RoboDK station: DalsySinBD.rdk

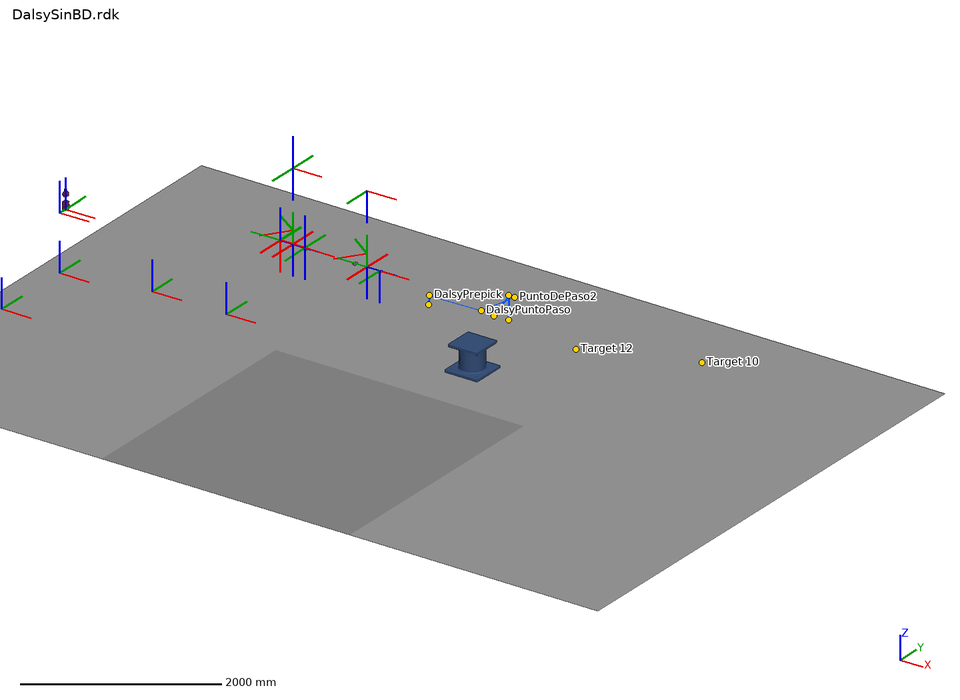
[picture v0: the station drawn from its stored meshes, robots at their saved joint values, targets as dots, program paths as lines]
Station EstacionProyectoFinaleliminarBotela (saved by RoboDK 5.9.4). Poses are relative to the parent item; angles as X-Y-Z fixed-axis rotations.
Station parameters (name, value as stored): Posicion, [[ 2850.000 ]] , CantBot1, 0, NUMBOTELLA1, 0, ElimBotellas1, 0, detectado1, 0, repes1, 0, Prellena1, 0, Prellena, 0, Detectado1, 0, IO_5, 1, NewPick, 0, Pinza, 1, NewPlace, 0, waituntil Detectado1, 1, Ventosa_plegado_caja, 0, CantCaja, 1.0, SCajaInicial, 1, SCajaPlace, 0, if(SCajaInicial, SyntaxError: Unexpected token `=', If(SCajaInicial, SyntaxError: Unexpected token `=', Mesa, 1, Mesa1, 0, Mesa2, 0, Mesa3, 0, MesaE, 0, MesaS, 1, Temperatura, 0, SensorMqtt, 0, LotesPendientes, 1
  - folder ESTACIÓN
    - folder Suelo
      - object Floor at (4500, 1500, 0) mm, size 3000 x 3000 x 0 mm, geometry from Floor.sld
      - object Floor2 at (1500, 1500, 0) mm, size 3000 x 3000 x 0 mm, geometry from Floor.sld
      - object Floor3 at (1500, 4500, 0) mm, size 3000 x 3000 x 0 mm, geometry from Floor.sld
      - object Floor4 at (4500, 4500, 0) mm, size 3000 x 3000 x 0 mm, geometry from Floor.sld
      - object Floor6 at (7500, 1500, 0) mm, size 3000 x 3000 x 0 mm, geometry from Floor.sld
      - object Floor5 at (7500, 4500, 0) mm, size 3000 x 3000 x 0 mm, geometry from Floor.sld
    - folder Mesa Giratoria
  - frame SisGeneral at (0, -19.13, 0) mm
    - folder CintayRobot
      - frame SisRefPick at (250, 2217.22, 0) mm
        - frame Cinta Botellas 1 at (0, 1000, 0) mm
          - robot CintaUno: 1 axes
              modified DH rows (alpha deg, a mm, theta deg, d mm): 0, 0, 0, 0 linear
              base shift (0, 0, 0) mm, rotated rx 0 ry 90 rz 0 deg
              joint limits [0] to [4500]; home [0]; saved at [0]
            - frame FrameBotellaSave at (0, 0, 0) mm
              - object Guardado at (0, 0, 0) mm, size 71.4 x 71.4 x 222.2 mm, 1042852009 curves, geometry from Bottle-Label.sld
            - frame Move at (0, 0, 0) mm
              - frame FrameBotella at (0, 100, 0) mm
                - object botella0 at (0, 0, 0) mm, size 71.4 x 71.4 x 222.2 mm, 1039516303 curves, geometry from Bottle-Label.sld
          - target Inicio (Cartesian target) at (0, 100, 863) mm; joints [0] of CintaUno
          - target Final (Cartesian target) at (4325.5, 559.3, 913.95) mm, rotated rx -90 ry 0 rz 90 deg; joints [0, -90, -90, 0, 90, 0] of CintaUno
          - frame TANQUE 1 at (1750, -902.14, 647.6) mm
            - frame Cono at (1000, 1000, 1240) mm, rotated rx 180 ry 0 rz 0 deg
              - object Cone 500x500mm at (0, 0, 0) mm
            - frame Deposito at (1000, 1000, 1240) mm
              - object Deposito at (0, 0, 0) mm
            - frame Frame 24 at (1000.71, 1000.6, 551.36) mm, rotated rx 180 ry 0 rz -124.91 deg
              - object Cylinder 50x150mm at (0, 0, 0) mm
            - frame Frame 25 at (1000.71, 1000.6, 401.36) mm, rotated rx -180 ry 0 rz -90 deg
              - object Cylinder 50x150mm at (0, 0, 0) mm
            - frame Frame 26 at (1000.71, 1000.6, 401.36) mm, rotated rx 90 ry 0 rz 90 deg
              - object Cylinder 50x150mm at (0, 0, 0) mm
            - frame Frame 27 at (1150.71, 1000.6, 401.36) mm, rotated rx -180 ry 0 rz 0 deg
              - object Cylinder 50x150mm at (0, 0, 0) mm
            - frame Frame 25 at (1000.71, 1000.6, 401.36) mm, rotated rx -180 ry 0 rz -90 deg
              - object Cylinder 50x150mm at (0, 0, 0) mm
            - frame Frame 25 at (850.71, 1000.6, 401.36) mm, rotated rx -180 ry 0 rz -90 deg
              - object Cylinder 50x150mm at (0, 0, 0) mm
            - frame Frame 25 at (850.71, 1000.6, 401.36) mm, rotated rx 0 ry 90 rz 0 deg
              - object Cylinder 50x150mm at (0, 0, 0) mm
            - frame Frame 31 at (850.65, 1001.38, 406.13) mm
              - object Sphere D100mm at (0, 0, 0) mm, size 50 x 50 x 25 mm, 1060155569 curves, geometry from Sphere-D100mm.sld
            - frame Frame 31 at (1151.57, 999.51, 402.52) mm
              - object Sphere D100mm at (0, 0, 0) mm, size 50 x 50 x 25 mm, 1060155569 curves, geometry from Sphere-D100mm.sld
          - frame DispensaTapones at (2650, -902.14, 647.6) mm
            - frame Cono at (1000, 1000, 1240) mm, rotated rx 180 ry 0 rz 0 deg
              - object Cone 500x500mm at (0, 0, 0) mm
            - frame Frame 24 at (1000.71, 1000.6, 551.36) mm, rotated rx 180 ry 0 rz -124.91 deg
              - object Cylinder 50x150mm at (0, 0, 0) mm
            - frame Frame 25 at (1000.71, 1000.6, 401.36) mm, rotated rx -180 ry 0 rz -90 deg
              - object Cylinder 50x150mm at (0, 0, 0) mm
            - frame Frame 26 at (1000.71, 1000.6, 401.36) mm, rotated rx 90 ry 0 rz 90 deg
              - object Cylinder 50x150mm at (0, 0, 0) mm
            - frame Frame 27 at (1150.71, 1000.6, 401.36) mm, rotated rx -180 ry 0 rz 0 deg
              - object Cylinder 50x150mm at (0, 0, 0) mm
            - frame Frame 25 at (1000.71, 1000.6, 401.36) mm, rotated rx -180 ry 0 rz -90 deg
              - object Cylinder 50x150mm at (0, 0, 0) mm
            - frame Frame 25 at (850.71, 1000.6, 401.36) mm, rotated rx -180 ry 0 rz -90 deg
              - object Cylinder 50x150mm at (0, 0, 0) mm
            - frame Frame 25 at (850.71, 1000.6, 401.36) mm, rotated rx 0 ry 90 rz 0 deg
              - object Cylinder 50x150mm at (0, 0, 0) mm
            - frame Frame 31 at (850.65, 1001.38, 406.13) mm
              - object Sphere D100mm at (0, 0, 0) mm, size 50 x 50 x 25 mm, 1060155569 curves, geometry from Sphere-D100mm.sld
            - frame Frame 31 at (1151.57, 999.51, 402.52) mm
              - object Sphere D100mm at (0, 0, 0) mm, size 50 x 50 x 25 mm, 1060155569 curves, geometry from Sphere-D100mm.sld
          - frame Sensor3 at (3498.8, -14.22, 715.35) mm, rotated rx 0 ry 0 rz 88.62 deg
            - object B2 at (0, 0, 0) mm
          - frame Sensor2 at (4402.28, -29.98, 715.35) mm, rotated rx 0 ry 0 rz 88.62 deg
            - object B1 at (0, 0, 0) mm
          - frame Sensor1 at (2598.8, -14.22, 715.35) mm, rotated rx 0 ry 0 rz 88.62 deg
            - object B0 at (0, 0, 0) mm
          - target DalsyPrepick (Cartesian target) at (4404.64, 97.25, 945.23) mm, rotated rx -179.46 ry -0.56 rz 92.6 deg; joints [67.794, -102.103, -28.32, -139.861, 89.279, 65.196] of UR5PickDalsy
          - target DalsyPick (Cartesian target) at (4400.29, 94.49, 846.14) mm, rotated rx -179.46 ry -0.56 rz 92.6 deg; joints [67.407, -90.716, -60.305, -119.258, 89.278, 64.809] of UR5PickDalsy
          - target DalsyPuntoPaso (Cartesian target) at (4989.54, 154.84, 921.17) mm, rotated rx 176.54 ry 3.78 rz 107.72 deg; joints [150.48, -91.95, -47.39, -125.54, 89.98, 132.65] of UR5PickDalsy
          - target PuntoDePaso2 (Cartesian target) at (5091.93, 592.06, 921.34) mm, rotated rx 176.53 ry 3.81 rz 169.24 deg; joints [212.01, -91.94, -47.38, -125.53, 89.97, 132.65] of UR5PickDalsy
          - target PrePlace (Cartesian target) at (5051.88, 544.46, 950.34) mm, rotated rx 179.87 ry 0 rz -95.46 deg; joints [208.979, -92.535, -38.825, -138.744, 90.075, 34.439] of UR5PickDalsy
          - target Place (Cartesian target) at (5051.88, 544.46, 680.34) mm, rotated rx 179.87 ry 0 rz -95.46 deg; joints [208.979, -74.687, -99.618, -95.799, 90.075, 34.439] of UR5PickDalsy
          - target Target 9 (Cartesian target) at (5079.28, 251.73, 846.24) mm, rotated rx -179.45 ry -0.55 rz -167.69 deg; joints [167.11, -90.71, -60.3, -119.25, 89.27, 64.8] of UR5PickDalsy
          - target Target 10 (Cartesian target) at (7103.35, 957.35, 614.14) mm, rotated rx -138.15 ry 89.07 rz -48.26 deg; joints [177.195, -131.024, -49.86, -164.778, 177.217, -76.295]
          - target Target 11 (Cartesian target) at (4404.64, 97.25, 945.23) mm, rotated rx -179.46 ry -0.56 rz 92.6 deg; joints [67.794, -102.103, -28.32, -139.861, 89.279, 65.196] of UR5PickDalsy
          - target Target 12 (Cartesian target) at (5875.13, 535.29, 591.77) mm, rotated rx -124.69 ry 88.93 rz 144.57 deg; joints [23.154, -118.729, -72.709, -170.068, 203.904, -92.258]
        - frame UR5 BasePickDalsy at (4673.46, 1459.5, 355) mm, rotated rx 0 ry 0 rz 180 deg
          - robot UR5PickDalsy (model UR5): 6 axes
              modified DH rows (alpha deg, a mm, theta deg, d mm): 0, 0, 0, 89.2; 90, 0, 180, 0; 0, 425, 0, 0; 0, 392, 0, 109.3; -90, 0, 0, 94.75; 90, 0, 180, 82.5
              joint limits [-360, -360, -360, -360, -360, -360] to [360, 360, 360, 360, 360, 360]; home [0, -90, -90, 0, 90, 0]; saved at [67.794, -102.103, -28.32, -139.861, 89.279, 65.196]
            - tool GripperPick, TCP at (0, 0, 130) mm
            - tool GripperPickV, TCP at (0, 0, 130) mm
          - frame Frame 45 at (4.13, 0, -300) mm
            - object Pedestal R1 at (0, 0, 0) mm, size 400 x 400 x 304.8 mm, 1065353216 curves, geometry from Pedestal-H12in-Type-1.sld
      - folder ProgramasDeLaCinta
        - Python program AvanzaCinta1 (listed below)
        - Python program AvanzaCinta2 (listed below)
        - Python program ResetBot (listed below)
        - program ProgCinta1 (11 instructions, listed below)
        - Python program ProgCintaUno (listed below)
      - folder Sensores
        - Python program ProgB0 (listed below)
        - Python program ProgB1 (listed below)
        - Python program ProgB2 (listed below)
      - folder ProgramasUr
        - program DalsyPickPlace (33 instructions, listed below)
        - Python program PickDalsy (listed below)
        - Python program PlaceDalsy (listed below)
        - Python program BorrarBotella (listed below)
    - folder Mesa
      - frame MesaGiratoriaBase at (5724.13, 3717.02, 0) mm
        - robot MesaGiratoria: 1 axes
            modified DH rows (alpha deg, a mm, theta deg, d mm): 0, 0, 0, 0
            joint limits [-200] to [200]; home [0]; saved at [110]
          - frame SistMesaGiratoria at (0, 1000, 0) mm
          - frame Place_caja at (-410, 300, 573) mm, rotated rx 0 ry 0 rz -40 deg
            - object cajaplace1.0 at (310.2, 492.2, 15.02) mm, rotated rx 0 ry 0 rz -70 deg
        - folder ScriptsMesa
          - Python program MoverMesa (listed below)
          - program MoverMesaBucle (3 instructions, listed below)
        - object Sensor_place_caja at (-90, -30, 510) mm, rotated rx 0 ry 0 rz -90 deg
        - object SensorDetectaCajaSalida at (-100, -10, 510) mm
  - folder PROGRAMA_PRINCIPAL
    - program Main (9 instructions, listed below)
  - folder MQTT
    - Python program mqttlistener (listed below)
    - Python program RobotController (listed below)
    - folder BaseDeDatos
      - Python program ConsultarBD (listed below)
      - Python program CrearBotellaBD (listed below)
      - Python program LlenarBD (listed below)
      - Python program ResetBD (listed below)
      - Python program EmpaquetarBD (listed below)
      - Python program TaponarBD (listed below)
    - folder JugarBD
      - Python program CrearLotesBD (listed below)
      - Python program TerminarLotesBD (listed below)
  - Python program RobotPickAndPlace (listed below)
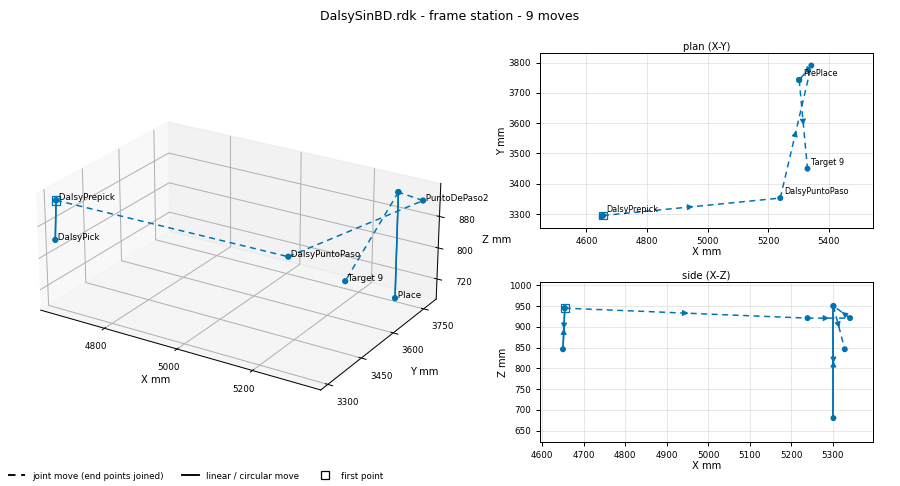
[picture p0: tool path of DalsySinBD.rdk in frame station, 9 of 9 moves have a stored position in this frame; points joined in program order, loops and branches not executed]

--- Python program AvanzaCinta1 ---
# Type help("robodk.robolink") or help("robodk.robomath") for more information
# Press F5 to run the script
# Documentation: https://robodk.com/doc/en/RoboDK-API.html
# Reference:     https://robodk.com/doc/en/PythonAPI/robodk.html
# Note: It is not required to keep a copy of this file, your Python script is saved with your RDK project

# You can also use the new version of the API:
from robodk import robolink    # RoboDK API
from robodk import robomath    # Robot toolbox
from robodk import time
RDK = robolink.Robolink()


cinta=RDK.Item('CintaUno')
INCREMENTO_MM=50

botella=RDK.Item('Bot')
Posicion1=cinta.Joints().list()


botella.setColor([0.47, 0.27, 0.08, 1])
while Posicion1[0]<2899.0000:
    if cinta.Valid():
        RDK.setParam('Posicion',cinta.Joints())
        cinta.MoveJ(cinta.Joints()+INCREMENTO_MM)
    Posicion1=cinta.Joints().list()

botella.setColor([1.0, 0.55, 0.63, 1])
while Posicion1[0]<4500.0000:
    if cinta.Valid():
        RDK.setParam('Posicion',cinta.Joints())
        cinta.MoveJ(cinta.Joints()+INCREMENTO_MM)
    Posicion1=cinta.Joints().list()

--- Python program AvanzaCinta2 ---
# Type help("robodk.robolink") or help("robodk.robomath") for more information
# Press F5 to run the script
# Documentation: https://robodk.com/doc/en/RoboDK-API.html
# Reference:     https://robodk.com/doc/en/PythonAPI/robodk.html
# Note: It is not required to keep a copy of this file, your Python script is saved with your RDK project

# You can also use the new version of the API:
from robodk import robolink    # RoboDK API
from robodk import robomath    # Robot toolbox
from robodk import time
RDK = robolink.Robolink()


cinta=RDK.Item('CintaSalidas')
INCREMENTO_MM=50


Posicion1=cinta.Joints().list()



while Posicion1[0]<2899.0000:
    if cinta.Valid():
        RDK.setParam('Posicion',cinta.Joints())
        cinta.MoveJ(cinta.Joints()+INCREMENTO_MM)
    Posicion1=cinta.Joints().list()

--- Python program ResetBot ---
from robodk import robolink
from robodk import robomath

RDK = robolink.Robolink()

# VARIABLES INICIALES
PonCero = 0

NUMBOTELLA = int(RDK.getParam('NUMBOTELLA1') or 0)
Eliminadas = 0  # Empezamos desde 0

# BORRAR TODAS LAS BOTELLAS DINÁMICAS
for i in range(NUMBOTELLA+1):
    botella = RDK.Item(f'botella{i}')
    if botella.Valid() and "Save" not in botella.Name():
        botella.Delete()
    Eliminadas += 1
botella = RDK.Item(f'botella{0.0}')
#botella.Delete()

# RESET PARAMS
RDK.setParam('CantBot1', PonCero)
RDK.setParam('NUMBOTELLA1', PonCero)
RDK.setParam('ElimBotellas1', PonCero)
RDK.setParam('repes1', PonCero)
RDK.setParam('Prellena1', PonCero)
RDK.setParam('Detectado1', PonCero)
RDK.setParam('NewPick', PonCero)
RDK.setParam('NewPlace', PonCero)

RDK.setParam('Mesa', 1)
RDK.setParam('MesaE', 1)
RDK.setParam('MesaS', 1)
RDK.setParam('Mesa1', 0)
RDK.setParam('Mesa2', 0)
RDK.setParam('Mesa3', 1)

# RESETEAR CINTA Y FRAME
cinta = RDK.Item('CintaUno')
Move = RDK.Item('Move')

if cinta.Valid():
    cinta.setJoints([50])

if Move.Valid():
    Move.setPose(robomath.transl(0, 0, 0))

# CREAR LA PRIMERA BOTELLA
BotellaBase = RDK.Item('Guardado')
FrameBotella = RDK.Item('FrameBotella')
color_granate_marron = [0.50, 0.12, 0.12, 1.0]

if BotellaBase.Valid() and FrameBotella.Valid():
    BotellaBase.Copy()
    botellaNueva = RDK.Paste(FrameBotella)
    botellaNueva.setName("botella0.0")
    botellaNueva.setVisible(True)
    botellaNueva.setColor(color_granate_marron)

--- program ProgCinta1 (robot CintaUno) ---
  while Detectado1==0
  if Prellena1==0
  while Temperatura == 1
  Pausa 500 ms
  end
  Llamar ProgCintaUno
  end
  if Prellena1!=0
  Pausa 5 ms
  end
  end

--- Python program ProgCintaUno ---
# Type help("robodk.robolink") or help("robodk.robomath") for more information
# Press F5 to run the script
# Documentation: https://robodk.com/doc/en/RoboDK-API.html
# Reference: https://robodk.com/doc/en/PythonAPI/robodk.html
# Note: It is not required to keep a copy of this file, your Python script is saved with your RDK project

# You can also use the new version of the API:
# Press F5 to run the script
# Documentation: https://robodk.com/doc/en/RoboDK-API.html
# Reference: https://robodk.com/doc/en/PythonAPI/robodk.html

from robodk import robolink    # RoboDK API
from robodk import robomath    # Robot toolbox

RDK = robolink.Robolink()

INCREMENTO_MM = 150

cinta = RDK.Item('CintaUno')
Botella = RDK.Item('botella0.0')
Guardado = RDK.Item('Guardado')
SisRef = RDK.Item('FrameBotella')
Move = RDK.Item('Move')

repes = RDK.getParam('repes1')

if cinta.Valid():

    NUMBOTELLA = RDK.getParam('NUMBOTELLA1')
    NUMBOTELLA += 1

    pose_actual = Move.Pose()
    nueva_pose = pose_actual

    pose = cinta.Pose()
    x_actual = pose[0, 3]

    if x_actual >= 4200:
        cinta.setJoints([0])
        repes = repes + 1
        Move.setPose(robomath.transl(x_actual * repes, 0, 0))
        RDK.setParam('repes1', repes)

    cinta.MoveJ(cinta.Joints() + INCREMENTO_MM)

    Guardado.Copy()
    GuardadoCopia = RDK.Paste(SisRef)
    GuardadoCopia.setName(f'botella{NUMBOTELLA}')

    CantBot = RDK.getParam('CantBot1')
    CantBot += 1

    GuardadoCopia.setPose(robomath.transl(-INCREMENTO_MM * CantBot, 0, 0))

    # GuardadoCopia.setPose(Botella.Pose() * robomath.transl(-INCREMENTO_MM * CantBot))

    GuardadoCopia.setVisible(True)

    RDK.setParam('CantBot1', CantBot)
    RDK.setParam('NUMBOTELLA1', NUMBOTELLA)

--- Python program ProgB0 ---
from robodk import robolink
from robodk import robomath

RDK = robolink.Robolink()

Sensor = RDK.Item('B0')

Inicio2 = 0
estadodetectado = 0
cuenta = 0

color_rosa_dalsy = [1.0, 0.75, 0.8, 1.0]

botella = RDK.Item(f'botella{Inicio2}')

while True:

    detectado = 1 if botella.Valid() and Sensor.Collision(botella) else 0

    if detectado != estadodetectado:

        if detectado == 1:
            cuenta += 1

            if cuenta == 3:
                cuenta = 0

                # pintar las 3 últimas botellas
                for i in range(3):
                    pinta = RDK.Item(f'botella{Inicio2 - i}')
                    if pinta.Valid():
                        pinta.setColor(color_rosa_dalsy)

        else:
            if cuenta < 3:
                RDK.setParam('Prellena1', 0)

        estadodetectado = detectado

        # avanzar a la siguiente botella
        if detectado == 0:
            Inicio2 += 1
            botella = RDK.Item(f'botella{Inicio2}')

    robomath.pause(0.01)

--- Python program ProgB1 ---
from robodk import robolink
from robodk import robomath
import paho.mqtt.client as mqtt

RDK = robolink.Robolink()

# MQTT config
broker = "broker.emqx.io"
port = 1883
user = "giiroB22"
passwd = "UPV2024"
station_status_topic = "giirob/pr2/station/mesa/status"

client = mqtt.Client()
client.username_pw_set(user, passwd)
client.connect(broker, port, 60)

Sensor = RDK.Item('B1')

inicio1 = 0
estadodetectado = 0
cuenta = 0

botella = RDK.Item(f'botella{inicio1}')

while True:

    if botella.Valid():
        detectado = 1 if Sensor.Collision(botella) else 0
    else:
        detectado = 0

    if detectado != estadodetectado:

        if detectado == 1:
            RDK.setParam('Detectado1', 1)
            RDK.setParam('Prellena1', 1)
            cuenta += 1

            # 📡 Publicar MQTT
            client.publish(station_status_topic, "sensor_detecta")
            print("[MQTT] sensor_detecta")

        else:
            RDK.setParam('Detectado1', 0)

            # 📡 Publicar MQTT
            client.publish(station_status_topic, "sensor_no_detecta")
            print("[MQTT] sensor_no_detecta")

            # avanzar a siguiente botella
            inicio1 += 1
            botella = RDK.Item(f'botella{inicio1}')

        estadodetectado = detectado

    # si no existe la botella, avanzar igualmente
    if not botella.Valid():
        inicio1 += 1
        botella = RDK.Item(f'botella{inicio1}')

    robomath.pause(0.01)

--- Python program ProgB2 ---
from robodk import robolink
from robodk import robomath

RDK = robolink.Robolink()

Sensor = RDK.Item('B2')

Inicio2 = 0
estadodetectado = 0
cuenta = 0

color_rosa_dalsy = [1.0, 0.9, 0.5, 1.0]

botella = RDK.Item(f'botella{Inicio2}')

while True:

    detectado = 1 if botella.Valid() and Sensor.Collision(botella) else 0

    if detectado != estadodetectado:

        if detectado == 1:
            cuenta += 1

            if cuenta == 3:
                cuenta = 0

                for i in range(3):
                    pinta = RDK.Item(f'botella{Inicio2 - i}')
                    if pinta.Valid():
                        pinta.setColor(color_rosa_dalsy)

        else:
            if cuenta < 3:
                RDK.setParam('Prellena1', 0)

        estadodetectado = detectado

        if detectado == 0:
            Inicio2 += 1
            botella = RDK.Item(f'botella{Inicio2}')

    robomath.pause(0.01)

--- program DalsyPickPlace (robot UR5PickDalsy) ---
  Est. Ref.: Cinta Botellas 1
  Est. herr: RobotiQ 2F-85 Gripper (Open) at (0, 0, 130) mm
  Set Pinza=0
  Establecer velocidad (700.0 mm/s)
  Pausa 500 ms
  while MesaE==0
  end
  MesaE=0
  while Detectado1==0
  MoveJ (DalsyPrepick)
  end
  Establecer velocidad (200.0 mm/s)
  MoveL (DalsyPick)
  Set Pinza=1
  Llamar PickDalsy
  Pausa 1.0 s
  MoveL (DalsyPrepick)
  Establecer velocidad (900.0 mm/s)
  MoveJ (DalsyPuntoPaso)
  Prellena1=0
  MoveJ (PuntoDePaso2)
  MoveJ (PrePlace)
  Establecer velocidad (200.0 mm/s)
  MoveL (Place)
  Llamar PlaceDalsy
  Set Pinza=1
  Llamar BorrarBotella
  Pausa 500 ms
  MoveL (PrePlace)
  Establecer velocidad (800.0 mm/s)
  MoveJ (Target 9)
  Pausa 1.0 s
  Mesa1=1

--- Python program PickDalsy ---
# Type help("robodk.robolink") or help("robodk.robomath") for more information
# Press F5 to run the script
# Documentation: https://robodk.com/doc/en/RoboDK-API.html
# Reference:     https://robodk.com/doc/en/PythonAPI/robodk.html
# Note: It is not required to keep a copy of this file, your Python script is saved with your RDK project

# You can also use the new version of the API:
from robodk import robolink    # RoboDK API
from robodk import robomath    # Robot toolbox
RDK = robolink.Robolink()

# Forward and backwards compatible use of the RoboDK API:
# Remove these 2 lines to follow python programming guidelines
from robodk import *      # RoboDK API
from robolink import *

# índice entero
new_pick = int(RDK.getParam('NewPick') or 0)

# límite de botellas creadas
max_botellas = int(RDK.getParam('NUMBOTELLA1') or 0)

# no avanzar si no existe aún
if new_pick >= max_botellas:
    quit()

botella = RDK.Item(f'botella{new_pick}')

robot = RDK.Item('GripperPick')
robot2 = RDK.Item('GripperPickV')

if botella.Valid() and robot.Valid():

    robot.DetachAll()
    robot.AttachClosest()

    new_pick += 1
    RDK.setParam('NewPick', new_pick)

    robot.setVisible(False)
    robot2.setVisible(True)

--- Python program PlaceDalsy ---
# Type help("robodk.robolink") or help("robodk.robomath") for more information
# Press F5 to run the script
# Documentation: https://robodk.com/doc/en/RoboDK-API.html
# Reference:     https://robodk.com/doc/en/PythonAPI/robodk.html

from robodk import robolink    # RoboDK API
from robodk import robomath    # Robot toolbox
from robodk import *
from robolink import *

RDK = robolink.Robolink()

# === Obtener índice global ===
new_Place = RDK.getParam('NewPlace')

# === Obtener botella por índice ===
botella = RDK.Item(f'botella{int(new_Place)}')

# === Obtener robot ===
robot = RDK.Item('GripperPick')  # <-- usa el nombre EXACTO del robot en RoboDK
robot2 = RDK.Item('GripperPickV')

# === Obtener sistema de coordenadas MesaGiratoria ===
mesa = RDK.Item('SistMesaGiratoria')   # <<< AÑADIDO

# === Verificación básica ===
if botella.Valid() and robot.Valid() and mesa.Valid():
    gripper = RDK.Item('GripperPick')


    # Obtener hijos (objetos cogidos)
    hijos = gripper.Childs()

    if len(hijos) > 0:
        objeto = hijos[0]
        if objeto.Valid():
            objeto.Delete()
    # === Soltar objeto del robot ===
    #robot.DetachAll()

    # === Mantener posición absoluta antes de cambiar parent ===
    #pose_abs = botella.PoseAbs()                     # <<< AÑADIDO

    # === Meter la botella en MesaGiratoria ===

    #botella.setParentStatic(mesa)
    #botella.setParent(mesa)                           # <<< AÑADIDO
    #botella.setPoseAbs(pose_abs)
    #botella.setPose(robomath.transl(0, 0, -9000))                  # <<< AÑADIDO

    # === Incrementar índice ===
    new_Place += 1
    RDK.setParam('NewPlace', new_Place)
    robot2.setVisible(False)   # Robot invisible
    robot.setVisible(True)

--- Python program BorrarBotella ---
from robodk.robolink import Robolink, ITEM_TYPE_OBJECT

RDK = Robolink()

# Obtener la ventosa
gripper = RDK.Item('GripperPick')


    # Obtener hijos (objetos cogidos)
hijos = gripper.Childs()

if len(hijos) > 0:
    objeto = hijos[0]

    if objeto.Valid():
        objeto.Delete()

--- Python program MoverMesa ---
# Type help("robodk.robolink") or help("robodk.robomath") for more information
# Press F5 to run the script
# Documentation: https://robodk.com/doc/en/RoboDK-API.html
# Reference:     https://robodk.com/doc/en/PythonAPI/robodk.html
# Note: It is not required to keep a copy of this file, your Python script is saved with your RDK project

# You can also use the new version of the API:
from robodk import robolink    # RoboDK API
from robodk import robomath
from robodk.robolink import Robolink

# Robot toolbox
RDK = Robolink()
import time

mesa=RDK.Item('MesaGiratoria')
sisRef=RDK.Item('Place_caja')
if mesa.Valid():
    giro=mesa.Joints().list()

    if( (giro[0]-90) <  (-200) ):
        giro[0] = 200
        for i in range(0,9):
            giro[0] = giro[0] - 10
            mesa.setJoints(giro)
            time.sleep(0.1)
    else:

        for i in range(0,9):
            giro[0] = giro[0]  -10
            mesa.setJoints(giro)
            time.sleep(0.1)



RDK.setParam('MesaE', 1)
RDK.setParam('Mesa1', 0)

--- program MoverMesaBucle (robot UR5PickDalsy) ---
  if Mesa1==1
  Llamar MoverMesa
  end

--- program Main (robot UR5PickDalsy) ---
  Llamar ResetBot
  Ejecutar ProgB0
  Ejecutar ProgB1
  Ejecutar ProgB2
  Ejecutar ProgCinta1
  Ejecutar RobotPickAndPlace
  Ejecutar MoverMesaBucle
  Ejecutar mqttlistener
  Ejecutar ResetBD

--- Python program mqttlistener ---
#from robodk import robolink    # RoboDK API
#from robodk import robomath    # Robot toolbox
#RDK = robolink.Robolink()

#import paho.mqtt.client as mqtt
#import RobotController as rc

#import paho.mqtt.client as mqtt
#import RobotController as rc

#broker="broker.emqx.io"
#port=1883
#user="giirob222"
#passwd="UPV2024"
#base_topic="giirob/pr2/station/"
#station_name="demo"
#station_commands_topic="giirob/pr2/station/mesa/commands"
#station_status_topic="giirob/pr2/station/mesa/status"

#def on_message(mqttc, obj, msg):
#    payload = msg.payload.decode('utf-8')
#    topic = msg.topic
#    qos = msg.qos
#    rc.handle_message(mqttc, topic, payload)

#mqttc = mqtt.Client(mqtt.CallbackAPIVersion.VERSION2)
#mqttc.on_message = on_message
#mqttc.username_pw_set(username=user, password=passwd)
#mqttc.connect(broker, port, 60)
#mqttc.subscribe(station_commands_topic, 0)
#mqttc.publish(station_status_topic)
#mqttc.loop_forever()

from robodk import robolink
import paho.mqtt.client as mqtt
import RobotController as rc  # Importamos nuestro controlador

# Configuración MQTT
broker = "broker.emqx.io"#mqtt.dsic.upv.es/broker.emqx.io
port = 1883
user = "giiroB22"
passwd = "UPV2024"
station_commands_topic = "giirob/pr2/station/mesa/commands"
station_status_topic = "giirob/pr2/station/mesa/status"

# Función que se ejecuta al recibir un mensaje
def on_message(client, userdata, msg):
    payload = msg.payload.decode('utf-8')
    topic = msg.topic
    print(f"[MQTT] Recibido: '{payload}' en topic: '{topic}'")
    rc.handle_message(topic, payload)  # solo topic y payload

# Crear cliente MQTT
client = mqtt.Client()
client.username_pw_set(user, passwd)
client.on_message = on_message

# Conectar al broker y suscribirse al topic de comandos
client.connect(broker, port, 60)
client.subscribe(station_commands_topic)

# Publicar status inicial
client.publish(station_status_topic, "online")
print("[MQTT] Publicado status: online")

# Bucle principal
client.loop_forever()

--- Python program RobotController ---
from robodk import robolink
RDK = robolink.Robolink()

variables = {
    "Temperatura": 0,
    "SensorMqtt": 0
}

def set_robodk_variable(name, value):
    try:
        RDK.setParam(name, str(value))
        print(f"[RoboDK] {name} = {value}")
    except Exception as e:
        print(f"ERROR: {e}")


def handle_message(topic, payload):

    payload = payload.strip()

    # -------------------------
    # TEMPERATURA
    # -------------------------
    if payload == "Temperatura_alta":
        variables["Temperatura"] = 1

    elif payload == "Temperatura_correcta":
        variables["Temperatura"] = 0

    # -------------------------
    # SENSOR MQTT
    # -------------------------
    elif payload == "SensorMqtt":
        variables["SensorMqtt"] = 1

    elif payload == "NotSensorMqtt":
        variables["SensorMqtt"] = 0

    else:
        print(f"[Controller] No reconocido: {payload}")
        return

    # -------------------------
    # DEBUG
    # -------------------------
    print(f"[Controller] Temperatura = {variables['Temperatura']}")
    print(f"[Controller] SensorMqtt = {variables['SensorMqtt']}")

    # -------------------------
    # UPDATE ROBO DK
    # -------------------------
    set_robodk_variable("Temperatura", variables["Temperatura"])
    set_robodk_variable("SensorMqtt", variables["SensorMqtt"])

--- Python program ConsultarBD ---
from robodk.robolink import *
import psycopg2
import time

RDK = Robolink()

conn = psycopg2.connect(
    host="127.0.0.1",
    database="postgres",
    user="postgres",
    password="30082004Aa",
    port="5432"
)

cur = conn.cursor()

print("Sistema iniciado")

while True:
    try:
        cur.execute("""
            SELECT COUNT(*)
            FROM lote
            WHERE estado IN ('pendiente', 'proceso')
        """)

        cantidad = cur.fetchone()[0]

        print("Cantidad:", cantidad)

        if cantidad > 0:
            RDK.setParam('LotesPendientes', '1')
        else:
            RDK.setParam('LotesPendientes', '0')


        RDK.Render()

    except Exception as e:
        print("Error:", e)
        RDK.setParam('LotesPendientes', '0')

    time.sleep(1)

--- Python program CrearBotellaBD ---
import psycopg2

conn = psycopg2.connect(
    host="127.0.0.1",
    database="postgres",
    user="postgres",
    password="30082004Aa",
    port="5432"
)

cur = conn.cursor()

cur.execute("""
    SELECT id
    FROM lote
    WHERE estado IN ('pendiente', 'proceso')
    ORDER BY id
    LIMIT 1
""")

resultado = cur.fetchone()

print("Resultado lote:", resultado)

if resultado:

    lote_id = resultado[0]

    cur.execute("""
        INSERT INTO botellas (
            llenada,
            taponada,
            empaquetada,
            lote_id
        )
        VALUES (FALSE, FALSE, FALSE, %s)
    """, (lote_id,))

    conn.commit()

    print("Botella insertada")

else:
    print("No hay lote disponible")

cur.close()
conn.close()

--- Python program LlenarBD ---
import psycopg2

conn = psycopg2.connect(
    host="127.0.0.1",
    database="postgres",
    user="postgres",
    password="30082004Aa",
    port="5432"
)

cur = conn.cursor()

# 1. Buscar 3 primeras botellas NO llenadas
cur.execute("""
    SELECT codigo
    FROM botellas
    WHERE llenada = FALSE
    ORDER BY codigo
    LIMIT 3
""")

botellas = cur.fetchall()

print("Botellas seleccionadas:", botellas)

# 2. Si hay botellas, marcarlas como llenadas
if len(botellas) > 0:

    for b in botellas:
        cur.execute("""
            UPDATE botellas
            SET llenada = TRUE
            WHERE codigo = %s
        """, (b[0],))

    conn.commit()

    print(" Bloque de llenado ejecutado")

else:
    print(" No hay botellas disponibles")

cur.close()
conn.close()

--- Python program ResetBD ---
import psycopg2

conn = psycopg2.connect(
    host="127.0.0.1",
    database="postgres",
    user="postgres",
    password="30082004Aa",
    port="5432"
)

cur = conn.cursor()

print(" Iniciando RESET completo...")

try:
    # 1. Borrar botellas
    cur.execute("DELETE FROM botellas;")
    print("✔ Botellas eliminadas")

    # 2. Borrar lotes
    cur.execute("DELETE FROM lote;")
    print("✔ Lotes eliminados")

    # 3. Reiniciar IDs (SERIAL)
    cur.execute("ALTER SEQUENCE botellas_codigo_seq RESTART WITH 1;")
    print("✔ Secuencia botellas reiniciada")

    cur.execute("ALTER SEQUENCE lote_id_seq RESTART WITH 1;")
    print("✔ Secuencia lotes reiniciada")

    conn.commit()

    print(" RESET COMPLETO FINALIZADO")

except Exception as e:
    print(" Error durante reset:", e)
    conn.rollback()

finally:
    cur.close()
    conn.close()

--- Python program EmpaquetarBD ---
import psycopg2

conn = psycopg2.connect(
    host="127.0.0.1",
    database="postgres",
    user="postgres",
    password="30082004Aa",
    port="5432"
)

cur = conn.cursor()

print("🔍 Buscando botella para empaquetar...")

try:
    # 1. Buscar primera botella lista para empaquetar
    cur.execute("""
        SELECT codigo
        FROM botellas
        WHERE llenada = TRUE
        AND empaquetada = FALSE
        ORDER BY codigo
        LIMIT 1
    """)

    botella = cur.fetchone()

    if botella:

        codigo = botella[0]

        # 2. Marcar como empaquetada
        cur.execute("""
            UPDATE botellas
            SET empaquetada = TRUE
            WHERE codigo = %s
        """, (codigo,))

        conn.commit()

        print(f"Botella {codigo} empaquetada")

    else:
        print(" No hay botellas listas para empaquetar")

except Exception as e:
    print(" Error:", e)
    conn.rollback()

finally:
    cur.close()
    conn.close()

--- Python program TaponarBD ---
import psycopg2

conn = psycopg2.connect(
    host="127.0.0.1",
    database="postgres",
    user="postgres",
    password="30082004Aa",
    port="5432"
)

cur = conn.cursor()

# 1. Buscar 3 primeras botellas NO llenadas
cur.execute("""
    SELECT codigo
    FROM botellas
    WHERE Taponada = FALSE
    ORDER BY codigo
    LIMIT 3
""")

botellas = cur.fetchall()

print("Botellas seleccionadas:", botellas)

# 2. Si hay botellas, marcarlas como llenadas
if len(botellas) > 0:

    for b in botellas:
        cur.execute("""
            UPDATE botellas
            SET Taponada = TRUE
            WHERE codigo = %s
        """, (b[0],))

    conn.commit()

    print(" Bloque de llenado ejecutado")

else:
    print(" No hay botellas disponibles")

cur.close()
conn.close()

--- Python program CrearLotesBD ---
import psycopg2

conn = psycopg2.connect(
    host="127.0.0.1",
    database="postgres",
    user="postgres",
    password="30082004Aa",
    port="5432"
)

cur = conn.cursor()

print(" Creando nuevo lote...")

try:
    cur.execute("""
        INSERT INTO lote (estado)
        VALUES ('pendiente')
    """)

    conn.commit()

    print(" Lote creado en estado PENDIENTE")

except Exception as e:
    print(" Error creando lote:", e)
    conn.rollback()

finally:
    cur.close()
    conn.close()

--- Python program TerminarLotesBD ---
import psycopg2
import time

conn = psycopg2.connect(
    host="127.0.0.1",
    database="postgres",
    user="postgres",
    password="30082004Aa",
    port="5432"
)

cur = conn.cursor()

print("Monitor de lotes iniciado...")

while True:
    try:
        # 1. Buscar lote activo
        cur.execute("""
            SELECT id
            FROM lote
            WHERE estado IN ('pendiente', 'proceso')
            ORDER BY id
            LIMIT 1
        """)

        lote = cur.fetchone()

        if lote:

            lote_id = lote[0]

            # 2. Contar empaquetadas del lote
            cur.execute("""
                SELECT COUNT(*)
                FROM botellas
                WHERE empaquetada = TRUE
                AND lote_id = %s
            """, (lote_id,))

            total = cur.fetchone()[0]

            print(f" Lote {lote_id} → {total}/30 empaquetadas")

            # 3. Si llega a 30 → cerrar lote
            if total >= 30:

                cur.execute("""
                    UPDATE lote
                    SET estado = 'terminado'
                    WHERE id = %s
                """, (lote_id,))

                conn.commit()

                print(f" LOTE {lote_id} TERMINADO")

        else:
            print(" No hay lote activo")

    except Exception as e:
        print("Error:", e)
        conn.rollback()

    time.sleep(1)

--- Python program RobotPickAndPlace ---
from robodk.robolink import *
import time

RDK = Robolink()

robot = RDK.Item('UR5PickDalsy')

if not robot.Valid():
    raise Exception("No se encontró el robot")

robot.setSpeed(700, 100)

while True:

    time.sleep(0.5)

    # Esperar MesaE
    while int(RDK.getParam("MesaE")) == 0:
        time.sleep(0.1)

    RDK.setParam("MesaE", 0)

    # Esperar detección
    DalsyPrepick = RDK.Item("DalsyPrepick")

    while int(RDK.getParam("SensorMqtt")) == 0:
        robot.MoveJ(DalsyPrepick)
        time.sleep(0.1)

    # bajar velocidad
    robot.setSpeed(200, 50)

    # PICK
    robot.MoveL(RDK.Item("DalsyPick"))

    PickDalsy = RDK.Item("PickDalsy")
    PickDalsy.RunProgram()
    PickDalsy.WaitFinished()

    time.sleep(1)

    robot.MoveL(DalsyPrepick)

    # subir velocidad
    robot.setSpeed(700, 100)

    robot.MoveJ(RDK.Item("DalsyPuntoPaso"))

    RDK.setParam("Prellena1", 0)

    robot.MoveJ(RDK.Item("PuntoDePaso2"))
    robot.MoveJ(RDK.Item("PrePlace"))

    robot.setSpeed(200, 50)

    robot.MoveL(RDK.Item("Place"))

    PlaceDalsy = RDK.Item("PlaceDalsy")
    PlaceDalsy.RunProgram()
    PlaceDalsy.WaitFinished()

    BorrarBotella = RDK.Item("BorrarBotella")
    BorrarBotella.RunProgram()
    BorrarBotella.WaitFinished()

    time.sleep(0.5)

    robot.MoveL(RDK.Item("PrePlace"))

    robot.setSpeed(700, 100)

    robot.MoveJ(RDK.Item("Target 9"))

    time.sleep(1)

    RDK.setParam("Mesa1", 1)
